(* IEC 61131-3 sources: teller/JD_Teller_LC2_V11/Class/Visu_Jam, 1 file *)

(* ---- Visu_Jam.st ---- *)
(*!
<Class
	Name               = "Visu_Jam"
	Revision           = "0.0"
	RealtimeTask       = "false"
	CyclicTask         = "false"
	BackgroundTask     = "true"
	Sigmatek           = "false"
	OSInterface        = "false"
	HighPriority       = "false"
	Automatic          = "false"
	UpdateMode         = "Prescan"
	SharedCommandTable = "true"
	Objectsize         = "(540,360)">
	<Channels>
		<Server Name="ClassSvr" Visualized="false" Initialize="false" WriteProtected="true" Retentive="false"/>
		<Server Name="JamBoxLength" Visualized="true" Initialize="false" WriteProtected="false" Retentive="false"/>
		<Server Name="oJamdetect" Visualized="false" Initialize="false" WriteProtected="true" Retentive="false"/>
		<Server Name="OnOff" Visualized="true" Initialize="false" WriteProtected="false" Retentive="false"/>
		<Server Name="oSensorHW" Visualized="true" Initialize="false" WriteProtected="true" Retentive="false"/>
		<Server Name="SensorNrInMachine" Visualized="true" Initialize="false" WriteProtected="false" Retentive="false"/>
		<Server Name="Status" Visualized="true" Initialize="false" WriteProtected="true" Retentive="false"/>
		<Server Name="TeachIn_Length" Visualized="true" Initialize="false" WriteProtected="true" Retentive="false"/>
		<Client Name="c_JamData" Required="true" Internal="false"/>
		<Client Name="c_SensorNr" Required="true" Internal="false"/>
	</Channels>
</Class>
*)
Visu_Jam : CLASS
  //Servers:
	ClassSvr 	: SvrChCmd_DINT;
	Status 	: SvrCh_tJamStatus;
	SensorNrInMachine 	: SvrCh_DINT;
	OnOff 	: SvrCh_DINT;
	oSensorHW 	: SvrCh_DINT;
	JamBoxLength 	: SvrCh_DINT;
	TeachIn_Length 	: SvrCh_DINT;
	oJamdetect 	: SvrCh_DINT;
  //Clients:
	c_JamData 	: CltChCmd_RAMex;
	c_SensorNr 	: CltCh_DINT;
  //Variables:
		JamData 	: ^tJamDetect;
  //Functions:

	FUNCTION VIRTUAL GLOBAL Init;

	FUNCTION VIRTUAL GLOBAL Background
		VAR_INPUT
			EAX 	: UDINT;
		END_VAR
		VAR_OUTPUT
			state (EAX) 	: UDINT;
		END_VAR;

	FUNCTION VIRTUAL GLOBAL Status::Read
		VAR_OUTPUT
			output (EAX) 	: tJamStatus;
		END_VAR;

	FUNCTION VIRTUAL GLOBAL SensorNrInMachine::Write
		VAR_INPUT
			input (EAX) 	: DINT;
		END_VAR
		VAR_OUTPUT
			result (EAX) 	: DINT;
		END_VAR;

	FUNCTION VIRTUAL GLOBAL OnOff::Write
		VAR_INPUT
			input (EAX) 	: DINT;
		END_VAR
		VAR_OUTPUT
			result (EAX) 	: DINT;
		END_VAR;

	FUNCTION VIRTUAL GLOBAL oSensorHW::Read
		VAR_OUTPUT
			output (EAX) 	: DINT;
		END_VAR;

	FUNCTION VIRTUAL GLOBAL JamBoxLength::Read
		VAR_OUTPUT
			output (EAX) 	: DINT;
		END_VAR;

	FUNCTION VIRTUAL GLOBAL JamBoxLength::Write
		VAR_INPUT
			input (EAX) 	: DINT;
		END_VAR
		VAR_OUTPUT
			result (EAX) 	: DINT;
		END_VAR;

	FUNCTION VIRTUAL GLOBAL TeachIn_Length::Read
		VAR_OUTPUT
			output (EAX) 	: DINT;
		END_VAR;
  //Tables:
	FUNCTION @STD
		VAR_OUTPUT
			ret_code	: CONFSTATES;
		END_VAR;
	FUNCTION GLOBAL TAB @CT_;
END_CLASS;

#pragma usingLtd RAMex

FUNCTION VIRTUAL GLOBAL Visu_Jam::Init

  if      c_JamData.GetSize() <> sizeof(tJamDetect) then
          c_JamData.SetSize(udSize:=sizeof(tJamDetect));
  end_if;

  if      _FirstScan then
          JamData := (c_JamData.GetDataPtr())$^tJamDetect;
          OnOff.Write(input:=JamData^.OnOff[c_SensorNr]);
          JamBoxLength.Write(input:=JamData^.JamBoxlength[c_SensorNr]);
          SensorNrInMachine.Write(input:=JamData^.SensorNrInMachine[c_SensorNr]);
  end_if;

END_FUNCTION

FUNCTION VIRTUAL GLOBAL Visu_Jam::Background
	VAR_INPUT
		EAX 	: UDINT;
	END_VAR
	VAR_OUTPUT
		state (EAX) 	: UDINT;
	END_VAR

  JamBoxLength.Read();
  TeachIn_Length.Read();
  Status.Read();
  oSensorHW.Read();

  if  Status = Jam_Detect then
      oJamdetect := 1;
  else
      oJamdetect := 0;
  end_if;

	state := READY;

END_FUNCTION

FUNCTION VIRTUAL GLOBAL Visu_Jam::Status::Read
	VAR_OUTPUT
		output (EAX) 	: tJamStatus;
	END_VAR

  Status :=  JamData^.Status[c_SensorNr];
	output := Status;

END_FUNCTION

FUNCTION VIRTUAL GLOBAL Visu_Jam::JamBoxLength::Read
	VAR_OUTPUT
		output (EAX) 	: DINT;
	END_VAR

  JamBoxLength := JamData^.JamBoxlength[c_SensorNr];
	output := JamBoxLength;

END_FUNCTION

FUNCTION VIRTUAL GLOBAL Visu_Jam::TeachIn_Length::Read
	VAR_OUTPUT
		output (EAX) 	: DINT;
	END_VAR

  TeachIn_Length := JamData^.TeachInLength[c_SensorNr];
	output := TeachIn_Length;

END_FUNCTION

FUNCTION VIRTUAL GLOBAL Visu_Jam::OnOff::Write
	VAR_INPUT
		input (EAX) 	: DINT;
	END_VAR
	VAR_OUTPUT
		result (EAX) 	: DINT;
	END_VAR

	OnOff := input;

  if OnOff < 0 | OnOff > 1 then
     OnOff := 0;
  end_if;

  JamData^.OnOff[c_SensorNr] := OnOff;
  if    JamData^.Status[c_SensorNr] = Turned_Off & JamBoxLength > 0 & OnOff then
        JamData^.Status[c_SensorNr] := Normal_Operation;
  elsif (JamData^.NrOfJamSensors >= c_SensorNr) & (JamBoxlength = 0 | OnOff = 0)  then
        JamData^.Status[c_SensorNr] := Turned_Off;
  end_if;

 	result := OnOff;

END_FUNCTION

FUNCTION VIRTUAL GLOBAL Visu_Jam::JamBoxLength::Write
	VAR_INPUT
		input (EAX) 	: DINT;
	END_VAR
	VAR_OUTPUT
		result (EAX) 	: DINT;
	END_VAR

	JamBoxLength := input;
  if    JamBoxLength < 0 then
        JamBoxLength := 0;
  elsif JamBoxLength > 2000 then    //eventueel aanpassen aan max t waarde boxeditor!!!!
        JamBoxLength := 2000;
  end_if;

  if    JamData^.Status[c_SensorNr] = Turned_Off & JamBoxLength > 0 & OnOff then
        JamData^.Status[c_SensorNr] := Normal_Operation;
  elsif (JamData^.NrOfJamSensors >= c_SensorNr) & (JamBoxlength = 0 | OnOff = 0)  then
        JamData^.Status[c_SensorNr] := Turned_Off;
  end_if;

  JamData^.JamBoxlength[c_SensorNr] := JamBoxLength;
 	result := JamBoxLength;

END_FUNCTION

FUNCTION VIRTUAL GLOBAL Visu_Jam::oSensorHW::Read
	VAR_OUTPUT
		output (EAX) 	: DINT;
	END_VAR

  oSensorHW := JamData^.Sensor[c_SensorNr];
	output := oSensorHW;

END_FUNCTION

FUNCTION VIRTUAL GLOBAL Visu_Jam::SensorNrInMachine::Write
	VAR_INPUT
		input (EAX) 	: DINT;
	END_VAR
	VAR_OUTPUT
		result (EAX) 	: DINT;
	END_VAR

	SensorNrInMachine := input;
  if  SensorNrInMachine < 0 then
      SensorNrInMachine := 0;
  elsif SensorNrInMachine > 100 then
        SensorNrInMachine := 100;
  end_if;
  JamData^.SensorNrInMachine[c_SensorNr] := SensorNrInMachine;

 	result := SensorNrInMachine;

END_FUNCTION
